// TIA Portal V17 export
// export: Created 2025-07-17T00:36:38.6791357Z, ExportSetting WithDefaults, DisplayName Totally Integrated Automation Portal, DisplayVersion V17, DisplayName TIA Portal Openness, DisplayVersion V17, DisplayName TIA Portal Version Control Interface, DisplayVersion V17, DisplayName STEP 7 Professional, DisplayVersion V17, DisplayName STEP 7 Safety, DisplayVersion V17, DisplayName WinCC Advanced / Unified PC, DisplayVersion V17
FUNCTION "RS-485_connect" : Void   // FC5, LAD
{ S7_Optimized_Access := 'TRUE' }
VERSION : 0.1
// stored: AutoNumber true, IsIECCheckEnabled false, SetENOAutomatically false, UDAEnableTagReadback false
   VAR_TEMP   // added for the SCL form of the ladder/FBD networks
      _w1 : Bool;
      _w2 : Bool;
      _w3 : Bool;
      _w4 : Bool;
      _w5 : Bool;
   END_VAR
BEGIN

REGION Network 1: 读从站
   // 读流量计从站
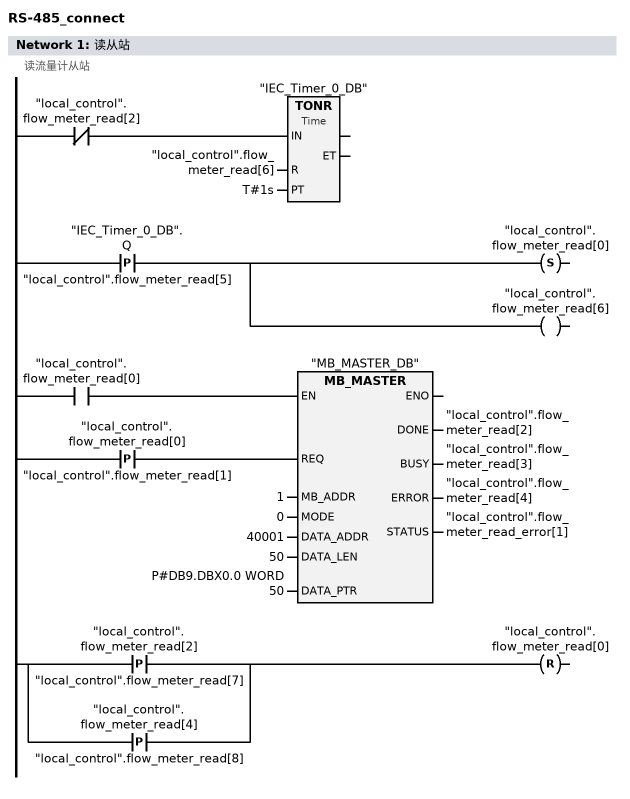
   RUNG wire#powerrail
      I_Contact( "local_control".flow_meter_read[2] )
      { S7_Templates := "time_type := Time" } "IEC_Timer_0_DB".TONR(r := "local_control".flow_meter_read[6], pt := T#1s, et =>)
   END_RUNG
   RUNG wire#powerrail
      P_Contact(operand := "IEC_Timer_0_DB".Q, bit := "local_control".flow_meter_read[5])
      wire#w1
      S_Coil( "local_control".flow_meter_read[0] )
   END_RUNG
   RUNG wire#w1
      Coil( "local_control".flow_meter_read[6] )
   END_RUNG
   RUNG wire#powerrail
      Contact( "local_control".flow_meter_read[0] )
      "MB_MASTER_DB".MB_MASTER(REQ := wire#w2, MB_ADDR := 1, MODE := 0, DATA_ADDR := 40001, DATA_LEN := 50, DATA_PTR := P#DB9.DBX0.0 WORD 50, DONE => "local_control".flow_meter_read[2], BUSY => "local_control".flow_meter_read[3], ERROR => "local_control".flow_meter_read[4], STATUS => "local_control".flow_meter_read_error[1])
   END_RUNG
   RUNG wire#powerrail
      P_Contact(operand := "local_control".flow_meter_read[0], bit := "local_control".flow_meter_read[1])
   END_RUNG wire#w2
   RUNG wire#powerrail
      P_Contact(operand := "local_control".flow_meter_read[2], bit := "local_control".flow_meter_read[7])
      wire#w3
      R_Coil( "local_control".flow_meter_read[0] )
   END_RUNG
   RUNG wire#powerrail
      P_Contact(operand := "local_control".flow_meter_read[4], bit := "local_control".flow_meter_read[8])
   END_RUNG wire#w3
   // the same network as SCL:
   "IEC_Timer_0_DB".TONR(IN := NOT "local_control".flow_meter_read[2],
                         R := "local_control".flow_meter_read[6],
                         PT := T#1s);
   #_w1 := "IEC_Timer_0_DB".Q AND NOT "local_control".flow_meter_read[5];   // rising edge of "IEC_Timer_0_DB".Q
   "local_control".flow_meter_read[5] := "IEC_Timer_0_DB".Q;
   IF #_w1 THEN "local_control".flow_meter_read[0] := TRUE; END_IF;
   "local_control".flow_meter_read[6] := #_w1;
   #_w3 := "local_control".flow_meter_read[0];
   #_w2 := "local_control".flow_meter_read[0] AND NOT "local_control".flow_meter_read[1];   // rising edge of "local_control".flow_meter_read[0]
   "local_control".flow_meter_read[1] := "local_control".flow_meter_read[0];
   IF #_w3 THEN
       "MB_MASTER_DB"(REQ := #_w2,   // MB_MASTER
                      MB_ADDR := 1,
                      MODE := 0,
                      DATA_ADDR := 40001,
                      DATA_LEN := 50,
                      DATA_PTR := P#DB9.DBX0.0 WORD 50,
                      DONE => "local_control".flow_meter_read[2],
                      BUSY => "local_control".flow_meter_read[3],
                      ERROR => "local_control".flow_meter_read[4],
                      STATUS => "local_control".flow_meter_read_error[1]);
   END_IF;
   #_w4 := "local_control".flow_meter_read[2] AND NOT "local_control".flow_meter_read[7];   // rising edge of "local_control".flow_meter_read[2]
   "local_control".flow_meter_read[7] := "local_control".flow_meter_read[2];
   #_w5 := "local_control".flow_meter_read[4] AND NOT "local_control".flow_meter_read[8];   // rising edge of "local_control".flow_meter_read[4]
   "local_control".flow_meter_read[8] := "local_control".flow_meter_read[4];
   IF #_w4 OR #_w5 THEN "local_control".flow_meter_read[0] := FALSE; END_IF;
END_REGION
END_FUNCTION
